// TwinCAT 3 PLC project UnitTest
// Title: Tc3_UnitTest
// Company: Zerlauth
// Author: Peter Zerlauth
// ProjectVersion: 0.0.2.9
// Description: Twincat 3 unit test library
// ProgramVersion: 3.1.4024.0
// libraries:
//   Tc2_Standard, * (Beckhoff Automation GmbH)
//   Tc2_System, * (Beckhoff Automation GmbH)
//   Tc2_Utilities, * (Beckhoff Automation GmbH)
//   Tc3_Module, * (Beckhoff Automation GmbH)
// project tree:
//   Assert/ E_AdsError.TcDUT (not stored), E_Assert.TcDUT (not stored), FB_Assert.TcPOU (not stored), I_Assert.TcIO (not stored)
//   Base/ E_Base.TcDUT (not stored), FB_Base.TcPOU (not stored), F_GetCycleTime.TcPOU (not stored), F_GetName.TcPOU (not stored), I_Base.TcIO (not stored)
//   List/Builder/ FB_StringBuilder.TcPOU (not stored), I_StringBuilder.TcIO (not stored)
//   List/Object/ I_Object.TcIO, FB_ListObject.TcPOU (not stored), I_ListObject.TcIO (not stored)
//   Logger/ E_LogLevel.TcDUT, FB_TcLogger.TcPOU (not stored), FB_Logger.TcPOU (not stored), I_Logger.TcIO (not stored), ST_LoggerSettings.TcDUT (not stored)
//   File/ FB_File.TcPOU (not stored), I_File.TcIO (not stored)
//   List/String/ FB_ListSTRING.TcPOU (not stored), I_ListSTRING.TcIO (not stored)
//   Property/ FB_Property.TcPOU (not stored), I_Property.TcIO (not stored)
//   Testcase/ E_Testcase.TcDUT (not stored), ST_Testcase.TcDUT (not stored)
//   Testsuites/ FB_Testsuites.TcPOU (not stored), I_Testsuites.TcIO (not stored), ST_TestsuitesOptions.TcDUT, ST_Testsuites.TcDUT (not stored)
//   Testsuite/ FB_Testsuite.TcPOU (not stored), I_Testsuite.TcIO, ST_Testsuite.TcDUT (not stored), ST_TestsuiteOptions.TcDUT (not stored)
// real-time tasks:
//   TASK PlcTask: cycle T#10ms, priority 20, ADS port 350

// ---- Logger/E_LogLevel.TcDUT
{attribute 'qualified_only'}
{attribute 'strict'}
TYPE E_LogLevel :
(
	Debug:=		0, 
    Info:= 		1, 
    Warning:= 	2, 
    Error:= 	3, 
    Critical:= 	4
);
END_TYPE

// ---- Testsuites/ST_TestsuitesOptions.TcDUT
TYPE ST_TestsuitesOptions :
STRUCT
	sFilePathName:		STRING(255):= 'C:\report.xml';		// as Property
END_STRUCT
END_TYPE

// ---- List/Object/I_Object.TcIO
INTERFACE I_Object EXTENDS __SYSTEM.IQueryInterface

END_INTERFACE

// ---- Testsuite/I_Testsuite.TcIO
INTERFACE I_Testsuite EXTENDS I_Base

PROPERTY PUBLIC P_File : String(255)
GET
END_GET
SET
END_SET
END_PROPERTY

PROPERTY PUBLIC P_List : I_ListSTRING
GET
END_GET
END_PROPERTY

PROPERTY PUBLIC P_Logger : I_Logger
GET
END_GET
SET
END_SET
END_PROPERTY

PROPERTY PUBLIC P_Options : reference to ST_TestsuiteOptions
GET
END_GET
END_PROPERTY

PROPERTY PUBLIC P_Parent : I_Testsuites
GET
END_GET
SET
END_SET
END_PROPERTY

PROPERTY PUBLIC P_Testcase : INT
GET
END_GET
END_PROPERTY

END_INTERFACE
